{attribute addProperty BoxType "EL2521-0000-1016"}
{attribute addProperty Id "Set_counter_doneAT %I*BOOL813Counter_underflowAT %I*BOOL814Counter_overflowAT %I*BOOL815Sync_ErrorAT %I*BOOL8132TxPDO_ToggleAT %I*BOOL819Counter_valueAT %I*UINT16217"}
{attribute addProperty CRC "3515788845"}
{attribute addProperty SizeInBites "56"}
{attribute addProperty SizeInBytes "7"}
TYPE ENC_Status_compact_D18EAE2D :
STRUCT
	{attribute addProperty Name "Set_counter_done"}
	Set_counter_done AT %I* : BOOL;
	{attribute addProperty Name "Counter_underflow"}
	Counter_underflow AT %I* : BOOL;
	{attribute addProperty Name "Counter_overflow"}
	Counter_overflow AT %I* : BOOL;
	{attribute addProperty Name "Sync_Error"}
	Sync_Error AT %I* : BOOL;
	{attribute addProperty Name "TxPDO_Toggle"}
	TxPDO_Toggle AT %I* : BOOL;
	{attribute addProperty Name "Counter_value"}
	Counter_value AT %I* : UINT;
END_STRUCT
END_TYPE

(* stored: Version 1.2.0.0, ProductVersion 3.1.4024.9
   DUT ENC_Status_compact_D18EAE2D: Id {bbfe7c4c-c272-4bbf-a9ef-a615d2cc52b3} *)
